// TIA Portal V19 export
FUNCTION_BLOCK "LOmacApcFr_Main"   // FB25, LAD
{ S7_Optimized_Access := 'TRUE' }
// stored: MemoryReserve 100, SetENOAutomatically false
   VAR_IN_OUT
      OmacInterface : "LMOmacApcFr_TypeInterface";
   END_VAR
   VAR
      instLPMLV30_UnitModeStateManager { S7_SetPoint := 'True'} : "LPMLV30_UnitModeStateManager";
      instLPMLV30_UnitModeStateTimes { S7_SetPoint := 'True'} : "LPMLV30_UnitModeStateTimes";
      instLOmacApcFr_CumulativeTimeSplitDINT { S7_SetPoint := 'True'} : "LOmacApcFr_CumulativeTimeSplitDINT";
   END_VAR
   VAR_TEMP
      tempLocalSC : Bool;   // State complete signal (one cycle)
   END_VAR
BEGIN

REGION Network 1: State Complete
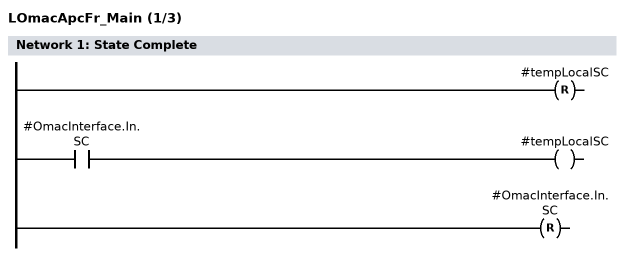
   RUNG wire#powerrail
      R_Coil( #tempLocalSC )
   END_RUNG
   RUNG wire#powerrail
      Contact( #OmacInterface.In.SC )
      Coil( #tempLocalSC )
   END_RUNG
   RUNG wire#powerrail
      R_Coil( #OmacInterface.In.SC )
   END_RUNG
   // the same network as SCL:
   #tempLocalSC := FALSE;
   #tempLocalSC := #OmacInterface.In.SC;
   #OmacInterface.In.SC := FALSE;
END_REGION

REGION Network 2: Call FB OMAC
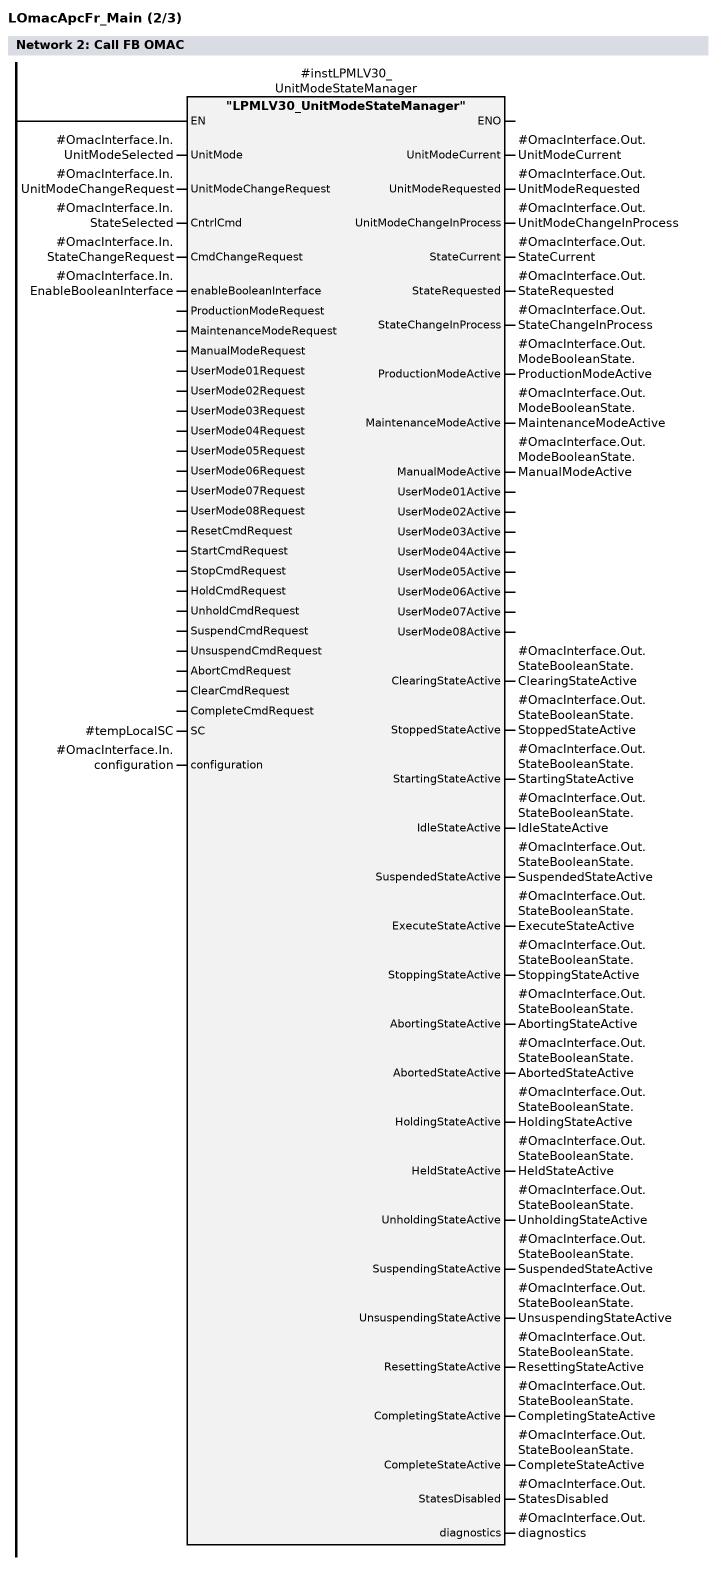
   RUNG wire#powerrail
      #instLPMLV30_UnitModeStateManager(UnitMode := #OmacInterface.In.UnitModeSelected, UnitModeChangeRequest := #OmacInterface.In.UnitModeChangeRequest, CntrlCmd := #OmacInterface.In.StateSelected, CmdChangeRequest := #OmacInterface.In.StateChangeRequest, enableBooleanInterface := #OmacInterface.In.EnableBooleanInterface, ProductionModeRequest :=, MaintenanceModeRequest :=, ManualModeRequest :=, UserMode01Request :=, UserMode02Request :=, UserMode03Request :=, UserMode04Request :=, UserMode05Request :=, UserMode06Request :=, UserMode07Request :=, UserMode08Request :=, ResetCmdRequest :=, StartCmdRequest :=, StopCmdRequest :=, HoldCmdRequest :=, UnholdCmdRequest :=, SuspendCmdRequest :=, UnsuspendCmdRequest :=, AbortCmdRequest :=, ClearCmdRequest :=, CompleteCmdRequest :=, SC := #tempLocalSC, configuration := #OmacInterface.In.configuration, UnitModeCurrent => #OmacInterface.Out.UnitModeCurrent, UnitModeRequested => #OmacInterface.Out.UnitModeRequested, UnitModeChangeInProcess => #OmacInterface.Out.UnitModeChangeInProcess, StateCurrent => #OmacInterface.Out.StateCurrent, StateRequested => #OmacInterface.Out.StateRequested, StateChangeInProcess => #OmacInterface.Out.StateChangeInProcess, ProductionModeActive => #OmacInterface.Out.ModeBooleanState.ProductionModeActive, MaintenanceModeActive => #OmacInterface.Out.ModeBooleanState.MaintenanceModeActive, ManualModeActive => #OmacInterface.Out.ModeBooleanState.ManualModeActive, UserMode01Active =>, UserMode02Active =>, UserMode03Active =>, UserMode04Active =>, UserMode05Active =>, UserMode06Active =>, UserMode07Active =>, UserMode08Active =>, ClearingStateActive => #OmacInterface.Out.StateBooleanState.ClearingStateActive, StoppedStateActive => #OmacInterface.Out.StateBooleanState.StoppedStateActive, StartingStateActive => #OmacInterface.Out.StateBooleanState.StartingStateActive, IdleStateActive => #OmacInterface.Out.StateBooleanState.IdleStateActive, SuspendedStateActive => #OmacInterface.Out.StateBooleanState.SuspendedStateActive, ExecuteStateActive => #OmacInterface.Out.StateBooleanState.ExecuteStateActive, StoppingStateActive => #OmacInterface.Out.StateBooleanState.StoppingStateActive, AbortingStateActive => #OmacInterface.Out.StateBooleanState.AbortingStateActive, AbortedStateActive => #OmacInterface.Out.StateBooleanState.AbortedStateActive, HoldingStateActive => #OmacInterface.Out.StateBooleanState.HoldingStateActive, HeldStateActive => #OmacInterface.Out.StateBooleanState.HeldStateActive, UnholdingStateActive => #OmacInterface.Out.StateBooleanState.UnholdingStateActive, SuspendingStateActive => #OmacInterface.Out.StateBooleanState.SuspendedStateActive, UnsuspendingStateActive => #OmacInterface.Out.StateBooleanState.UnsuspendingStateActive, ResettingStateActive => #OmacInterface.Out.StateBooleanState.ResettingStateActive, CompletingStateActive => #OmacInterface.Out.StateBooleanState.CompletingStateActive, CompleteStateActive => #OmacInterface.Out.StateBooleanState.CompleteStateActive, StatesDisabled => #OmacInterface.Out.StatesDisabled, diagnostics => #OmacInterface.Out.diagnostics)
   END_RUNG
   // the same network as SCL:
   #instLPMLV30_UnitModeStateManager(UnitMode := #OmacInterface.In.UnitModeSelected,   // "LPMLV30_UnitModeStateManager"
                           UnitModeChangeRequest := #OmacInterface.In.UnitModeChangeRequest,
                           CntrlCmd := #OmacInterface.In.StateSelected,
                           CmdChangeRequest := #OmacInterface.In.StateChangeRequest,
                           enableBooleanInterface := #OmacInterface.In.EnableBooleanInterface,
                           SC := #tempLocalSC,
                           configuration := #OmacInterface.In.configuration,
                           UnitModeCurrent => #OmacInterface.Out.UnitModeCurrent,
                           UnitModeRequested => #OmacInterface.Out.UnitModeRequested,
                           UnitModeChangeInProcess => #OmacInterface.Out.UnitModeChangeInProcess,
                           StateCurrent => #OmacInterface.Out.StateCurrent,
                           StateRequested => #OmacInterface.Out.StateRequested,
                           StateChangeInProcess => #OmacInterface.Out.StateChangeInProcess,
                           ProductionModeActive => #OmacInterface.Out.ModeBooleanState.ProductionModeActive,
                           MaintenanceModeActive => #OmacInterface.Out.ModeBooleanState.MaintenanceModeActive,
                           ManualModeActive => #OmacInterface.Out.ModeBooleanState.ManualModeActive,
                           ClearingStateActive => #OmacInterface.Out.StateBooleanState.ClearingStateActive,
                           StoppedStateActive => #OmacInterface.Out.StateBooleanState.StoppedStateActive,
                           StartingStateActive => #OmacInterface.Out.StateBooleanState.StartingStateActive,
                           IdleStateActive => #OmacInterface.Out.StateBooleanState.IdleStateActive,
                           SuspendedStateActive => #OmacInterface.Out.StateBooleanState.SuspendedStateActive,
                           ExecuteStateActive => #OmacInterface.Out.StateBooleanState.ExecuteStateActive,
                           StoppingStateActive => #OmacInterface.Out.StateBooleanState.StoppingStateActive,
                           AbortingStateActive => #OmacInterface.Out.StateBooleanState.AbortingStateActive,
                           AbortedStateActive => #OmacInterface.Out.StateBooleanState.AbortedStateActive,
                           HoldingStateActive => #OmacInterface.Out.StateBooleanState.HoldingStateActive,
                           HeldStateActive => #OmacInterface.Out.StateBooleanState.HeldStateActive,
                           UnholdingStateActive => #OmacInterface.Out.StateBooleanState.UnholdingStateActive,
                           SuspendingStateActive => #OmacInterface.Out.StateBooleanState.SuspendedStateActive,
                           UnsuspendingStateActive => #OmacInterface.Out.StateBooleanState.UnsuspendingStateActive,
                           ResettingStateActive => #OmacInterface.Out.StateBooleanState.ResettingStateActive,
                           CompletingStateActive => #OmacInterface.Out.StateBooleanState.CompletingStateActive,
                           CompleteStateActive => #OmacInterface.Out.StateBooleanState.CompleteStateActive,
                           StatesDisabled => #OmacInterface.Out.StatesDisabled,
                           diagnostics => #OmacInterface.Out.diagnostics);
END_REGION

REGION Network 3: Call FB Time Counter
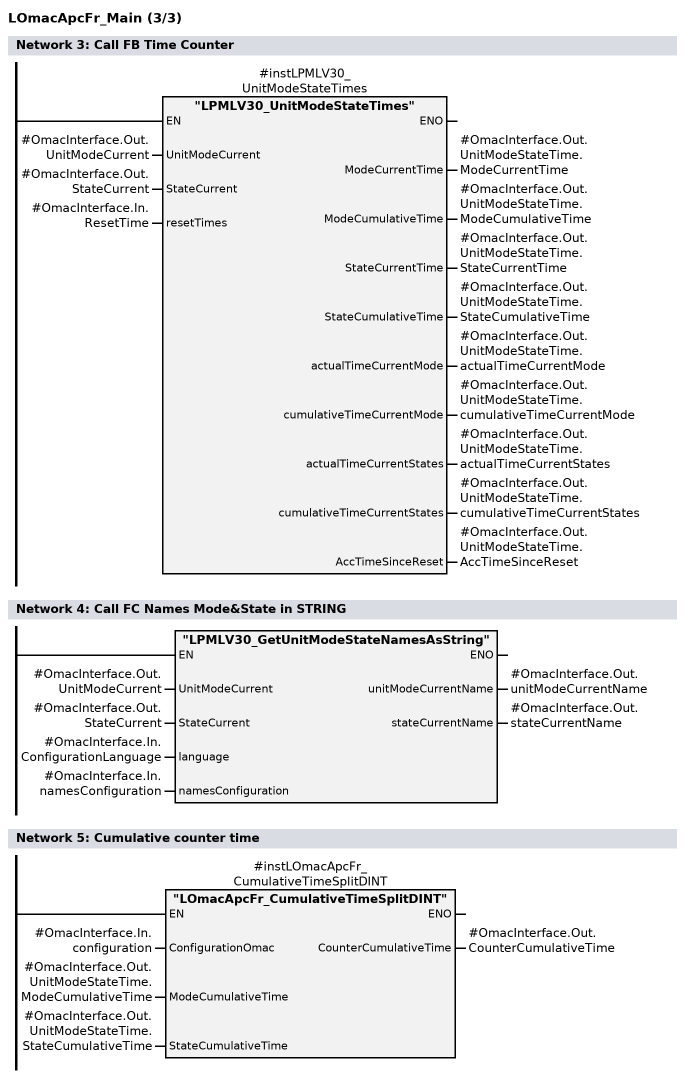
   RUNG wire#powerrail
      #instLPMLV30_UnitModeStateTimes(UnitModeCurrent := #OmacInterface.Out.UnitModeCurrent, StateCurrent := #OmacInterface.Out.StateCurrent, resetTimes := #OmacInterface.In.ResetTime, ModeCurrentTime => #OmacInterface.Out.UnitModeStateTime.ModeCurrentTime, ModeCumulativeTime => #OmacInterface.Out.UnitModeStateTime.ModeCumulativeTime, StateCurrentTime => #OmacInterface.Out.UnitModeStateTime.StateCurrentTime, StateCumulativeTime => #OmacInterface.Out.UnitModeStateTime.StateCumulativeTime, actualTimeCurrentMode => #OmacInterface.Out.UnitModeStateTime.actualTimeCurrentMode, cumulativeTimeCurrentMode => #OmacInterface.Out.UnitModeStateTime.cumulativeTimeCurrentMode, actualTimeCurrentStates => #OmacInterface.Out.UnitModeStateTime.actualTimeCurrentStates, cumulativeTimeCurrentStates => #OmacInterface.Out.UnitModeStateTime.cumulativeTimeCurrentStates, AccTimeSinceReset => #OmacInterface.Out.UnitModeStateTime.AccTimeSinceReset)
   END_RUNG
   // the same network as SCL:
   #instLPMLV30_UnitModeStateTimes(UnitModeCurrent := #OmacInterface.Out.UnitModeCurrent,   // "LPMLV30_UnitModeStateTimes"
                           StateCurrent := #OmacInterface.Out.StateCurrent,
                           resetTimes := #OmacInterface.In.ResetTime,
                           ModeCurrentTime => #OmacInterface.Out.UnitModeStateTime.ModeCurrentTime,
                           ModeCumulativeTime => #OmacInterface.Out.UnitModeStateTime.ModeCumulativeTime,
                           StateCurrentTime => #OmacInterface.Out.UnitModeStateTime.StateCurrentTime,
                           StateCumulativeTime => #OmacInterface.Out.UnitModeStateTime.StateCumulativeTime,
                           actualTimeCurrentMode => #OmacInterface.Out.UnitModeStateTime.actualTimeCurrentMode,
                           cumulativeTimeCurrentMode => #OmacInterface.Out.UnitModeStateTime.cumulativeTimeCurrentMode,
                           actualTimeCurrentStates => #OmacInterface.Out.UnitModeStateTime.actualTimeCurrentStates,
                           cumulativeTimeCurrentStates => #OmacInterface.Out.UnitModeStateTime.cumulativeTimeCurrentStates,
                           AccTimeSinceReset => #OmacInterface.Out.UnitModeStateTime.AccTimeSinceReset);
END_REGION

REGION Network 4: Call FC Names Mode&State in STRING
   RUNG wire#powerrail
      "LPMLV30_GetUnitModeStateNamesAsString"(UnitModeCurrent := #OmacInterface.Out.UnitModeCurrent, StateCurrent := #OmacInterface.Out.StateCurrent, language := #OmacInterface.In.ConfigurationLanguage, namesConfiguration := #OmacInterface.In.namesConfiguration, unitModeCurrentName => #OmacInterface.Out.unitModeCurrentName, stateCurrentName => #OmacInterface.Out.stateCurrentName)
   END_RUNG
   // the same network as SCL:
   "LPMLV30_GetUnitModeStateNamesAsString"(UnitModeCurrent := #OmacInterface.Out.UnitModeCurrent,
                           StateCurrent := #OmacInterface.Out.StateCurrent,
                           language := #OmacInterface.In.ConfigurationLanguage,
                           namesConfiguration := #OmacInterface.In.namesConfiguration,
                           unitModeCurrentName => #OmacInterface.Out.unitModeCurrentName,
                           stateCurrentName => #OmacInterface.Out.stateCurrentName);
END_REGION

REGION Network 5: Cumulative counter time
   RUNG wire#powerrail
      #instLOmacApcFr_CumulativeTimeSplitDINT(ConfigurationOmac := #OmacInterface.In.configuration, ModeCumulativeTime := #OmacInterface.Out.UnitModeStateTime.ModeCumulativeTime, StateCumulativeTime := #OmacInterface.Out.UnitModeStateTime.StateCumulativeTime, CounterCumulativeTime => #OmacInterface.Out.CounterCumulativeTime)
   END_RUNG
   // the same network as SCL:
   #instLOmacApcFr_CumulativeTimeSplitDINT(ConfigurationOmac := #OmacInterface.In.configuration,   // "LOmacApcFr_CumulativeTimeSplitDINT"
                           ModeCumulativeTime := #OmacInterface.Out.UnitModeStateTime.ModeCumulativeTime,
                           StateCumulativeTime := #OmacInterface.Out.UnitModeStateTime.StateCumulativeTime,
                           CounterCumulativeTime => #OmacInterface.Out.CounterCumulativeTime);
END_REGION
END_FUNCTION_BLOCK
